PROGRAM DatenRangieren
VAR	
	VersionsText: STRING := 'Labor Linearachse V2.0';
END_VAR

VersionsInfo.Ver := MAXSTRING_TO_BYTEARR(VersionsText);

IF VersionsInfo.Befehle = 16#00 THEN	// lokale Ein- und Ausgänge verwenden
	SimDI.ASCII := Plc_dSub.DI_LowByte;
	
	Plc_dSub.DQ_LowByte := AlleBitSetzen(	SimDa.P1R,
											SimDa.P1L,
											SimDa.P2R,
											SimDa.P2L,
											SimDa.P3R,	
											SimDa.P3L,	
											SimDa.P4R,	
											SimDa.P4L);	

	Plc_dSub.DQ_HighByte := AlleBitSetzen(	SimDa.P5R,
											SimDa.P5L,
											FALSE,
											FALSE,
											FALSE,	
											FALSE,	
											FALSE,	
											FALSE);										
ELSE	// Simulation (Digital Twin) verwenden	
	SimDI.ASCII := DigInput.DI[0];
	
	DigOutput.DA[0] := AlleBitSetzen(	SimDa.P1R,
											SimDa.P1L,
											SimDa.P2R,
											SimDa.P2L,
											SimDa.P3R,	
											SimDa.P3L,	
											SimDa.P4R,	
											SimDa.P4L);	
											
	DigOutput.DA[0] := AlleBitSetzen(		SimDa.P5R,
											SimDa.P5L,
											FALSE,
											FALSE,
											FALSE,	
											FALSE,	
											FALSE,	
											FALSE);											
END_IF

END_PROGRAM

(* stored: Version 1.1.0.1, ProductVersion 3.1.4024.4
   POU DatenRangieren: Id {ad49a684-d9e6-4dba-bece-08745f191ac1}, SpecialFunc None *)
